(* PLC project Unnamed, Unknown Unnamed 1 *)
(* stored: creationDateTime 2026-01-05T10:16:11, modificationDateTime 2026-01-05T10:16:11 *)

PROGRAM main
  VAR_INPUT
    X0 : BOOL;
  END_VAR
  VAR_OUTPUT
    Y0 : BOOL;
  END_VAR

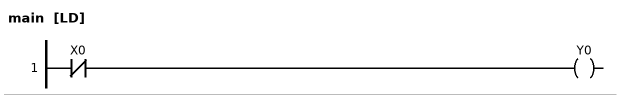
(* LD diagram, written out as Structured Text *)
Y0 := NOT X0;
END_PROGRAM

CONFIGURATION Config0
  RESOURCE Res0 ON PLC
    TASK task0(INTERVAL := T#20ms, PRIORITY := 1);
    PROGRAM instance0 WITH task0 : main;
  END_RESOURCE
END_CONFIGURATION
